(* IEC 61131-3 sources: ctf1-cps6963/plc1/build, 2 files *)

(* ---- plc.st ---- *)
TYPE
  LOGLEVEL : (CRITICAL, WARNING, INFO, DEBUG) := INFO;
END_TYPE

FUNCTION_BLOCK LOGGER
  VAR_INPUT
    TRIG : BOOL;
    MSG : STRING;
    LEVEL : LOGLEVEL := INFO;
  END_VAR
  VAR
    TRIG0 : BOOL;
  END_VAR

  IF TRIG AND NOT TRIG0 THEN
  {{
   LogMessage(GetFbVar(LEVEL),(char*)GetFbVar(MSG, .body),GetFbVar(MSG, .len));
  }}
  END_IF;
  TRIG0:=TRIG;
END_FUNCTION_BLOCK

PROGRAM plc1
  VAR
    ColorSensor_RED : INT;
    ColorSensor_GREEN : INT;
    ColorSensor_BLUE : INT;
    RangeSensor : INT;
    Pump : BOOL := False;
    treatmentComplete : BOOL := False;
  END_VAR
  VAR
    desiredDistanceFill : REAL := 7.0;
    measuredDistance : REAL;
  END_VAR

  (*Workaround to distance measure bug*)
  measuredDistance := INT_TO_REAL(RangeSensor)/100.0;
  desiredDistanceFill := 7.0;

  IF treatmentComplete THEN
          IF measuredDistance > desiredDistanceFill THEN
            Pump := TRUE;
          ELSE
            Pump := FALSE;
          END_IF;
  END_IF;
END_PROGRAM

CONFIGURATION Config0

  RESOURCE Res0 ON PLC
    TASK task0(INTERVAL := T#20ms,PRIORITY := 0);
    PROGRAM instance0 WITH task0 : plc1;
  END_RESOURCE
END_CONFIGURATION

(* ---- generated_plc.st ---- *)
PROGRAM plc1
  VAR
    ColorSensor_RED AT %IW0 : INT;
    ColorSensor_GREEN AT %IW1 : INT;
    ColorSensor_BLUE AT %IW2 : INT;
    RangeSensor AT %IW3 : INT;
    Pump AT %QX0.4 : BOOL := False;
    treatmentComplete AT %IX100.0 : BOOL := False;
  END_VAR
  VAR
    desiredDistanceFill : REAL := 7.0;
    measuredDistance : REAL;
  END_VAR

  (*Workaround to distance measure bug*)
  measuredDistance := INT_TO_REAL(RangeSensor)/100.0;
  desiredDistanceFill := 7.0;

  IF treatmentComplete THEN
          IF measuredDistance > desiredDistanceFill THEN
            Pump := TRUE;
          ELSE
            Pump := FALSE;
          END_IF;
  END_IF;
END_PROGRAM

CONFIGURATION Config0

  RESOURCE Res0 ON PLC
    TASK task0(INTERVAL := T#20ms,PRIORITY := 0);
    PROGRAM instance0 WITH task0 : plc1;
  END_RESOURCE
END_CONFIGURATION
